// TIA Portal V16 export
// export: Created 2026-06-18T08:11:22.6089421Z, ExportSetting WithDefaults, DisplayName Totally Integrated Automation Portal, DisplayVersion V16 Update 8, DisplayName TIA Portal Version Control Interface, DisplayVersion V16 Update 8, DisplayName TIA Portal Openness, DisplayVersion V16 Update 8, DisplayName SINAMICS Startdrive Advanced, DisplayVersion V16, DisplayName SINAMICS Startdrive G130, G150, S120, S150, SINAMICS MV, S210, DisplayVersion V16, DisplayName SINAMICS Startdrive G110M, G120, G120C, G120D, G120P, DisplayVersion V16, DisplayName STEP 7 Professional, DisplayVersion V16 Update 8, DisplayName STEP 7 Safety, DisplayVersion V16 Update 7, DisplayName WinCC Advanced, DisplayVersion V16 Update 8
Screen "Login_Screen"  800x480, Number=1
  ScreenLayer 
    IOField "IO_Password" at 430,280 size 240x44  DataFormat=Decimal, FormatPattern=9999999, Mode=InOutput
    Button "BTN_Login" at 430,380 size 130x54  Mode=Text, TextOff="登录", TextOn="登录"
    SymbolicIOField "符号 I/O 域_1" at 177,87 size 170x32  CountVisibleItems=3, Mode=InOutput, OnValue=1, TextOff="0", TextOn="1"
    Circle "LMP_Online" at 770,385 size 48x48
    TextField "TXT_OnlineStatus" at 810,395 size 80x36  Text="在线状态"
    Button "BTN_Logout" at 600,380 size 130x54  Mode=Text, TextOff="退出", TextOn="退出"
    Button "按钮_3" at 545,140 size 96x32  Mode=Text, TextOff="Text", TextOn="Text"
    Circle "圆_2" at 480,252 size 48x48
    Circle "圆_3" at 371,285 size 48x48
